// TIA Portal V17 export
// export: Created 2021-12-03T08:13:00.6031769Z, ExportSetting WithDefaults, DisplayName Totally Integrated Automation Portal, DisplayVersion V17, DisplayName TIA Portal Openness, DisplayVersion V17, DisplayName TIA Portal Version Control Interface, DisplayVersion V17, DisplayName STEP 7 Professional, DisplayVersion V17, DisplayName STEP 7 Safety, DisplayVersion V17, DisplayName WinCC Advanced, DisplayVersion V17
FUNCTION "FC_ScanSequence" : Void   // FC70, FBD
VERSION : 0.1
// stored: AutoNumber false, IsIECCheckEnabled false, UDAEnableTagReadback false
   VAR_TEMP
      T_ScanIntrrpt : Bool;
   END_VAR
BEGIN

REGION Network 1
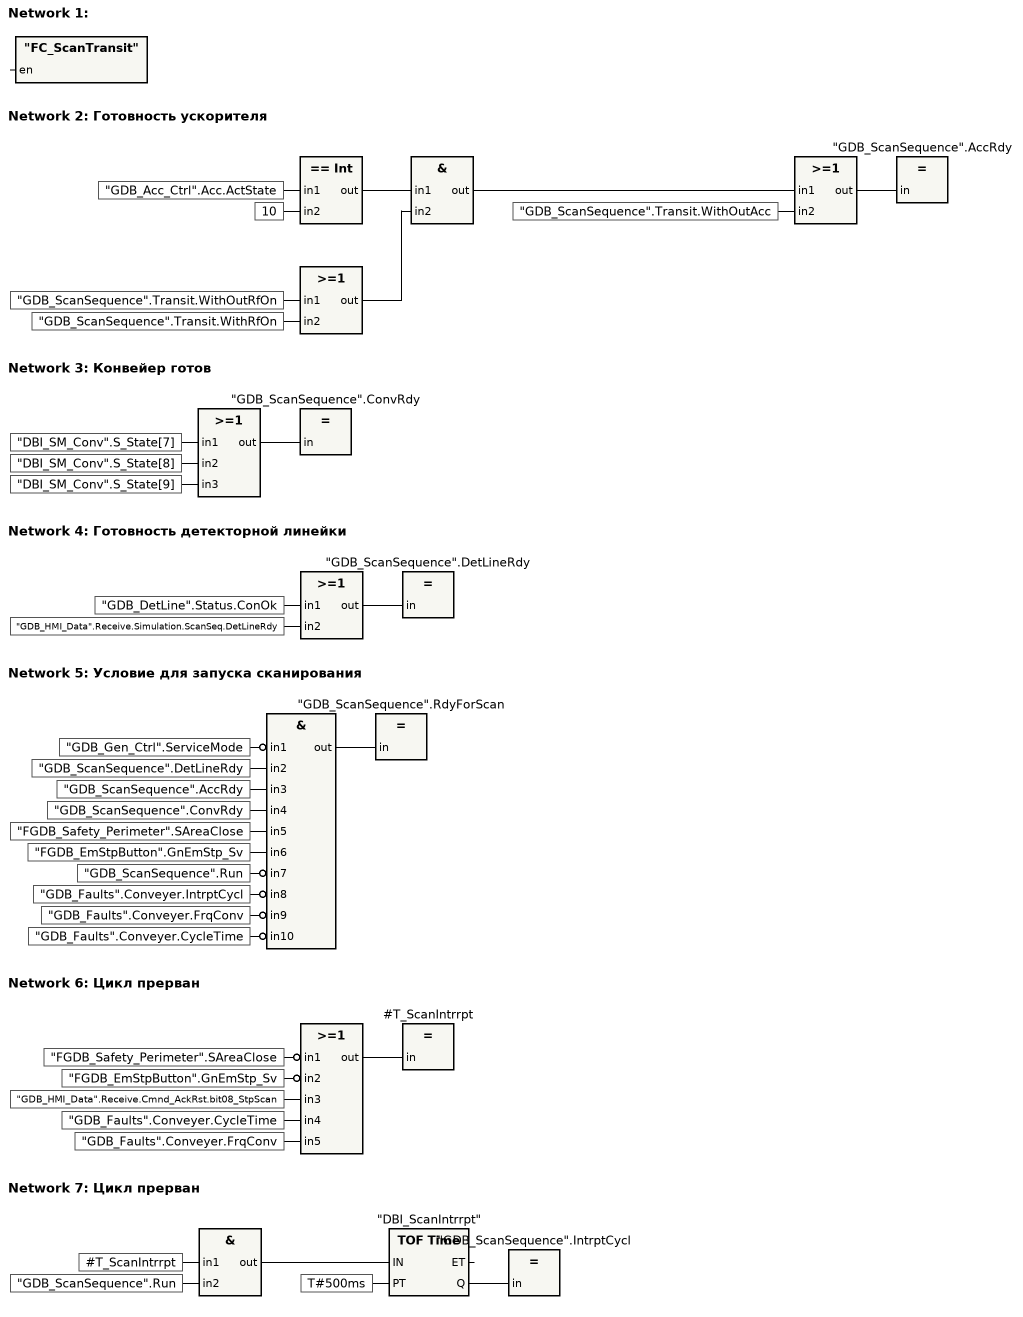
   "FC_ScanTransit"();
END_REGION

REGION Network 2: Готовность ускорителя
   "GDB_ScanSequence".AccRdy := (("GDB_Acc_Ctrl".Acc.ActState = 10) AND ("GDB_ScanSequence".Transit.WithOutRfOn OR "GDB_ScanSequence".Transit.WithRfOn)) OR "GDB_ScanSequence".Transit.WithOutAcc;
END_REGION

REGION Network 3: Конвейер готов
   "GDB_ScanSequence".ConvRdy := "DBI_SM_Conv".S_State[7] OR "DBI_SM_Conv".S_State[8] OR "DBI_SM_Conv".S_State[9];
END_REGION

REGION Network 4: Готовность детекторной линейки
   "GDB_ScanSequence".DetLineRdy := "GDB_DetLine".Status.ConOk OR "GDB_HMI_Data".Receive.Simulation.ScanSeq.DetLineRdy;
END_REGION

REGION Network 5: Условие для запуска сканирования
   "GDB_ScanSequence".RdyForScan := NOT "GDB_Gen_Ctrl".ServiceMode AND "GDB_ScanSequence".DetLineRdy AND "GDB_ScanSequence".AccRdy AND "GDB_ScanSequence".ConvRdy AND "FGDB_Safety_Perimeter".SAreaClose AND "FGDB_EmStpButton".GnEmStp_Sv AND NOT "GDB_ScanSequence".Run AND NOT "GDB_Faults".Conveyer.IntrptCycl AND NOT "GDB_Faults".Conveyer.FrqConv AND NOT "GDB_Faults".Conveyer.CycleTime;
END_REGION

REGION Network 6: Цикл прерван
   #T_ScanIntrrpt := NOT "FGDB_Safety_Perimeter".SAreaClose OR NOT "FGDB_EmStpButton".GnEmStp_Sv OR "GDB_HMI_Data".Receive.Cmnd_AckRst.bit08_StpScan OR "GDB_Faults".Conveyer.CycleTime OR "GDB_Faults".Conveyer.FrqConv;
END_REGION

REGION Network 7: Цикл прерван
   "DBI_ScanIntrrpt".TOF(IN := #T_ScanIntrrpt AND "GDB_ScanSequence".Run, PT := T#500ms);
   "GDB_ScanSequence".IntrptCycl := "DBI_ScanIntrrpt".Q;
END_REGION

REGION Network 8: Запуск сканирования
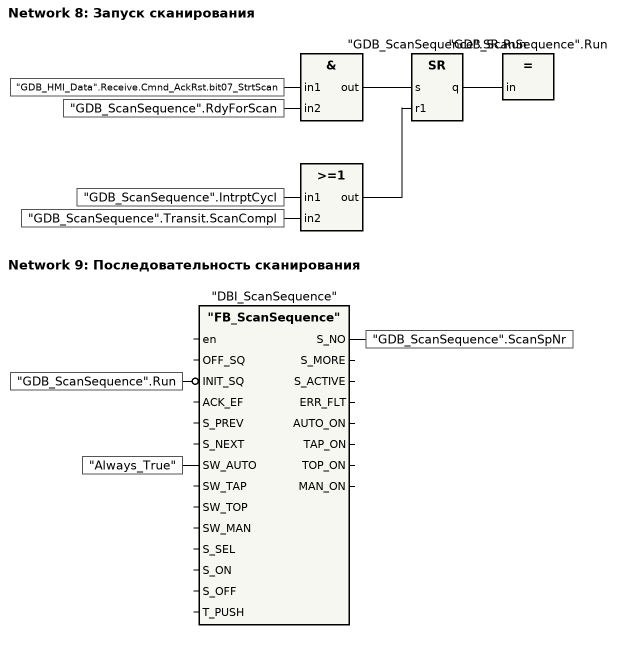
   IF "GDB_HMI_Data".Receive.Cmnd_AckRst.bit07_StrtScan AND "GDB_ScanSequence".RdyForScan THEN
       "GDB_ScanSequence".SR.Run := TRUE;   // SR flip-flop
   END_IF;
   IF "GDB_ScanSequence".IntrptCycl OR "GDB_ScanSequence".Transit.ScanCompl THEN
       "GDB_ScanSequence".SR.Run := FALSE;
   END_IF;
   "GDB_ScanSequence".Run := "GDB_ScanSequence".SR.Run;
END_REGION

REGION Network 9: Последовательность сканирования
   "DBI_ScanSequence"(INIT_SQ := NOT "GDB_ScanSequence".Run,   // "FB_ScanSequence"
                      SW_AUTO := "Always_True",
                      S_NO => "GDB_ScanSequence".ScanSpNr);
END_REGION
END_FUNCTION
